Staubli VAL3: JointTrajPtFMsg.pjx

--- JointTrajPtFMsg.pjx ---
Parameters version=s7.7.2 stackSize=5000 millimeterUnit=true
Program file=start.pgx
Program file=stop.pgx
Data file=JointTrajPtFMsg.dtx
Type name=Body path=Disk://Body/Body.pjx
Type name=Header path=Disk://Header/Header.pjx
Type name=Prefix path=Disk://Prefix/Prefix.pjx
Type name=JointTrajPtFull path=Disk://JointTrajPtFull/JointTrajPtFull.pjx

--- JointTrajPtFMsg.dtx ---
public Header header
  [0]
    num nMsgType
    num nCommType
    num nReplyCode
    num nData[12]
public Prefix prefix
  [0]
    num nLength
    num nData[4]
public JointTrajPtFull jointTrajPtFull
  [0]
    num nRobotId
    num nSeq
    num nValidFields
    num nTime
    num nPositions[10]
    num nVelocities[10]
    num nAccelerations[10]
public Body body
  [0]
    num nData[136]
